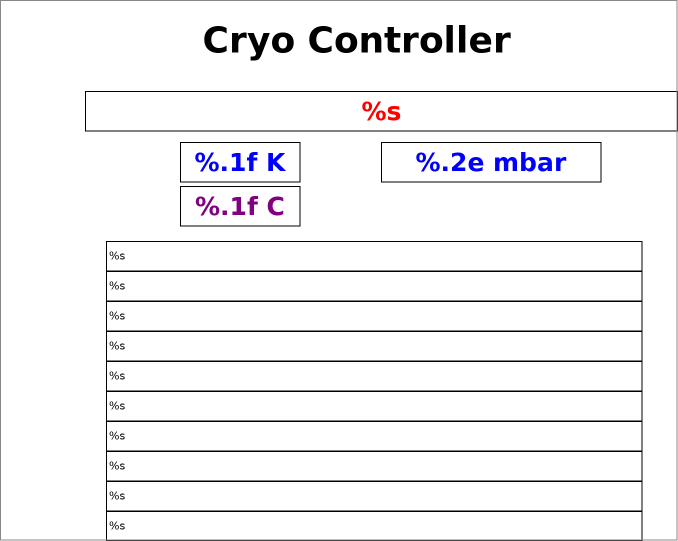
VISUALIZATION GUI_CRYO  // 678x541
    Rectangle (180,142 120x40), "%.1f K", text variable: MAIN.Cryo_Ctrl.Temp_ColdBench.stat.lrTempK
    Rectangle (180,186 120x40), "%.1f C", text variable: MAIN.Cryo_Ctrl.Temp_ColdBench.stat.lrTempC
    Rectangle (381,142 220x40), "%.2e mbar", text variable: MAIN.Cryo_Ctrl.Pressure_Cryo.stat.lrPressure
    Label (182,15 350x50), "Cryo Controller"
    Rectangle (85,91 593x40), "%s", text variable: MAIN.Cryo_Ctrl.stat.sState
    Rectangle (106,241 536x30), "%s", text variable: MAIN.Cryo_Ctrl.syslog.s9
    Rectangle (106,271 536x30), "%s", text variable: MAIN.Cryo_Ctrl.syslog.s8
    Rectangle (106,301 536x30), "%s", text variable: MAIN.Cryo_Ctrl.syslog.s7
    Rectangle (106,331 536x30), "%s", text variable: MAIN.Cryo_Ctrl.syslog.s6
    Rectangle (106,361 536x30), "%s", text variable: MAIN.Cryo_Ctrl.syslog.s5
    Rectangle (106,391 536x30), "%s", text variable: MAIN.Cryo_Ctrl.syslog.s4
    Rectangle (106,421 536x30), "%s", text variable: MAIN.Cryo_Ctrl.syslog.s3
    Rectangle (106,451 536x30), "%s", text variable: MAIN.Cryo_Ctrl.syslog.s2
    Rectangle (106,481 536x30), "%s", text variable: MAIN.Cryo_Ctrl.syslog.s1
    Rectangle (106,511 536x30), "%s", text variable: MAIN.Cryo_Ctrl.syslog.s0
END_VISUALIZATION

(* stored: Version 1.1.0.1, ProductVersion 3.1.4024.9
   Visu GUI_CRYO: Id {b7ef14d5-285a-446b-b24a-12a5d455d646} *)
